FUNCTION_BLOCK Pneumatic_1Coil_Management
// Function block untuk mengolah faceplate dan watchdog pneumatic valve 1 coil
//	UDT dependencies:
	(*  
	1. stPneumatic v1.0 	*)

//	Changelog:
	(* 
	v1.0 [27.12.2021] Start development function block - Fabrilian Asali	*)	

VAR_INPUT
	bEnable						: BOOL;		
	bTriggerPneumatic			: BOOL;
	bTestMode					: BOOL;
	bResetError					: BOOL;
	bBypassSensorRetract		: BOOL;
	bBypassSensorAdvanced		: BOOL;
	bBypassPreCheckSensor		: BOOL;
	xIn_SensorRetract			: BOOL;
	xIn_SensorAdvanced			: BOOL;
	TimerWatchdogRetract		: TIME := T#5S;
	TimerWatchdogAdvanced		: TIME := T#5S;
	TimerWatchdogPreRetract		: TIME := T#5S;
	TimerWatchdogPreAdvanced	: TIME := T#5S;
END_VAR

VAR_OUTPUT
	bError						: BOOL;
	ErrorID						: INT;
	ErrorMsg					: STRING;
END_VAR

VAR_IN_OUT
	Pneumatic					: stPneumatic1;
END_VAR

VAR
	SeqIndex					: INT;
	WatchdogTimer				: TON;
	bTrig_Output				: BOOL;
END_VAR
VAR // added by the converter: edge detectors and wires of the graphical bodies
    _rt1 : R_TRIG;
    _ft1 : F_TRIG;
END_VAR

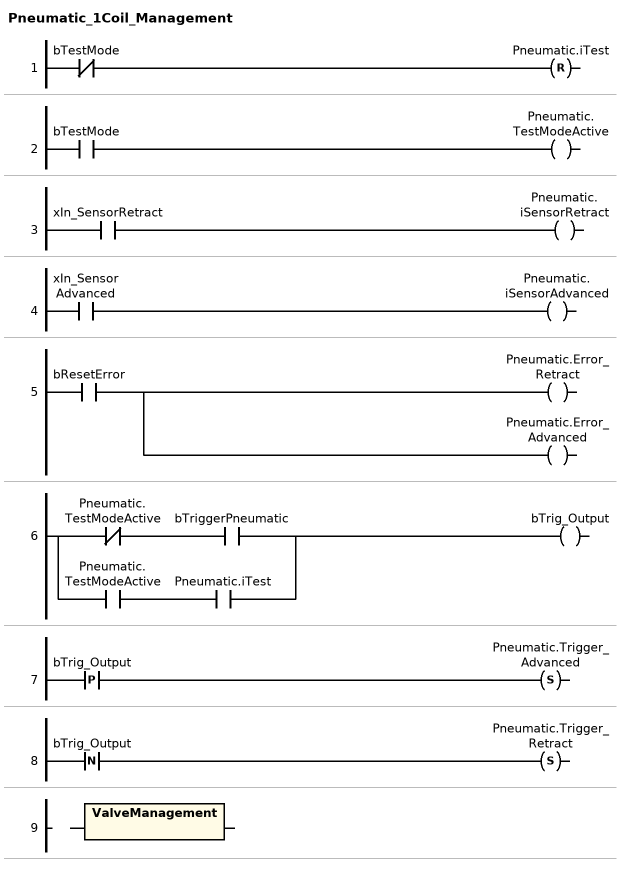
// NETWORK 1
Pneumatic.iTest R= NOT bTestMode;

// NETWORK 2
Pneumatic.TestModeActive := bTestMode;

// NETWORK 3
Pneumatic.iSensorRetract := xIn_SensorRetract;

// NETWORK 4
Pneumatic.iSensorAdvanced := xIn_SensorAdvanced;

// NETWORK 5
Pneumatic.Error_Retract := bResetError;
Pneumatic.Error_Advanced := bResetError;

// NETWORK 6
bTrig_Output := NOT Pneumatic.TestModeActive AND bTriggerPneumatic OR Pneumatic.TestModeActive AND Pneumatic.iTest;

// NETWORK 7
_rt1(CLK := bTrig_Output);
Pneumatic.Trigger_Advanced S= _rt1.Q;

// NETWORK 8
_ft1(CLK := bTrig_Output);
Pneumatic.Trigger_Retract S= _ft1.Q;

// NETWORK 9
ValveManagement();

ACTION ValveManagement:

IF bResetError THEN
	SeqIndex	:= 0;
	ErrorID		:= 0;
	ErrorMsg	:= '';
	bError		:= FALSE;
END_IF

IF bEnable AND NOT bError THEN
	CASE SeqIndex OF
		0:
			IF Pneumatic.Trigger_Retract THEN
				SeqIndex	:= 100;
			ELSIF Pneumatic.Trigger_Advanced THEN
				SeqIndex	:= 200;
			END_IF
		
		100:
			Pneumatic.Trigger_Retract	:= FALSE;
			IF NOT bBypassPreCheckSensor THEN
				WatchdogTimer(In:= TRUE, PT:= TimerWatchdogPreRetract);
				IF Pneumatic.iSensorAdvanced THEN
					WatchdogTimer(In:= FALSE);
					SeqIndex	:= 110;
				ELSIF WatchdogTimer.Q THEN
					WatchdogTimer(In:= FALSE);
					Pneumatic.Error_Retract := TRUE;
					ErrorID					:= 10;
					ErrorMsg				:= 'Error PreCheck Retract';
					SeqIndex	:= 999;
				END_IF
			ELSE
				SeqIndex	:= 110;
			END_IF
	
		110:
			Pneumatic.oPneumatic := FALSE;
			IF NOT bBypassSensorRetract THEN
				WatchdogTimer(In:= TRUE, PT:= TimerWatchdogRetract);
				IF Pneumatic.iSensorRetract THEN
					WatchdogTimer(In:= FALSE);
					SeqIndex	:= 0;
				ELSIF WatchdogTimer.Q THEN
					WatchdogTimer(In:= FALSE);
					Pneumatic.Error_Retract := TRUE;
					ErrorID					:= 11;
					ErrorMsg				:= 'Error Watchdog Retract';
				END_IF
			ELSE
				SeqIndex	:= 0;
			END_IF
			
		200:
			Pneumatic.Trigger_Advanced	:= FALSE;
			IF NOT bBypassPreCheckSensor THEN
				WatchdogTimer(In:= TRUE, PT:= TimerWatchdogPreAdvanced);
				IF Pneumatic.iSensorRetract THEN
					WatchdogTimer(In:= FALSE);
					SeqIndex	:= 210;
				ELSIF WatchdogTimer.Q THEN
					WatchdogTimer(In:= FALSE);
					Pneumatic.Error_Advanced := TRUE;
					ErrorID					:= 20;
					ErrorMsg				:= 'Error PreCheck Advanced';
					SeqIndex	:= 999;
				END_IF
			ELSE
				SeqIndex	:= 210;
			END_IF				
		
		210:
			Pneumatic.oPneumatic := TRUE;
			IF NOT bBypassSensorAdvanced THEN
				WatchdogTimer(In:= TRUE, PT:= TimerWatchdogAdvanced);
				IF Pneumatic.iSensorAdvanced THEN
					WatchdogTimer(In:= FALSE);
					SeqIndex	:= 0;
				ELSIF WatchdogTimer.Q THEN
					WatchdogTimer(In:= FALSE);
					Pneumatic.Error_Advanced := TRUE;
					ErrorID					:= 21;
					ErrorMsg				:= 'Error Watchdog Advanced';
				END_IF
			ELSE
				SeqIndex	:= 0;
			END_IF					
	
		999:
			bError	:= TRUE;	
			
	END_CASE
ELSE
	SeqIndex := 0;
	WatchdogTimer(IN:= FALSE);
	Pneumatic.Trigger_Advanced	:= FALSE;
	Pneumatic.Trigger_Retract	:= FALSE;
END_IF
END_ACTION

END_FUNCTION_BLOCK

(* stored: Version 1.1.0.1, ProductVersion 3.1.4024.9
   POU Pneumatic_1Coil_Management: Id {ccb4f153-69e5-4b35-b246-b531fd5cf5e3}, SpecialFunc None
   Action ValveManagement: Id {841fccbe-1ad3-4ca7-a1f5-b8b3ff32283d} *)
